// TIA Portal project "prova5arob" (V16)

(* hardware
DEVICE "S7-1200 station_1"  S7-1200 Station
   slot 0: "Telaio di montaggio_0"  S7-1200 Rack  Rack  V1.0
   slot 1: "PLC_1"  CPU 1215C DC/DC/Rly  6ES7 215-1HG40-0XB0  V4.2
DEVICE "HMI_1"  KTP700 Basic PN
   slot 0: "HMI_1"  KTP700 Basic PN  6AV2 123-2GB03-0AX0  16.0.0.0
   slot 1: "HMI_RT_1"  KTP700 Basic PN  6AV2 123-2GB03-0AX0  16.0.0.0
   slot 5: "HMI_1.IE_CP_1"  PROFINET Interface  16.0.0.0
      slot 1: "Interfaccia_1 PROFINET"  PROFINET Interface
         slot 1: "Porta_1"  Port
*)

// ===== PLC "PLC_1"  CPU 1215C DC/DC/Rly =====

DATA_BLOCK "Blocco_dati_pannello"   // DB1
{ S7_Optimized_Access := 'TRUE' }
VERSION : 0.1
   VAR
      Jog_start : Bool;
      spia_marcia : Bool;
   END_VAR
BEGIN
END_DATA_BLOCK

ORGANIZATION_BLOCK "Main"   // OB1, LAD, ProgramCycle
TITLE = "Main Program Sweep (Cycle)"
{ S7_Optimized_Access := 'TRUE' }
VERSION : 0.1
   VAR_INPUT
      Initial_Call : Bool;   // Initial call of this OB
      Remanence : Bool;   // =True, if remanent data are available
   END_VAR
BEGIN

REGION Network 1
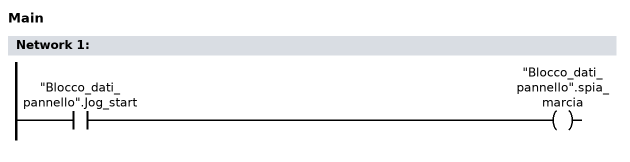
   RUNG wire#powerrail
      Contact( "Blocco_dati_pannello".Jog_start )
      Coil( "Blocco_dati_pannello".spia_marcia )
   END_RUNG
   // the same network as SCL:
   "Blocco_dati_pannello".spia_marcia := "Blocco_dati_pannello".Jog_start;
END_REGION
END_ORGANIZATION_BLOCK

(* ===== HMI "HMI_RT_1" =====
system functions are stored by id; their names below are inferred from use
connection "HMI_Collegamento_1": ETHERNET, SMART_S7_1200_OMS

HMI tags "Tabella delle variabili standard"
   "Variabile_Numero di pagina" : UInt, internal
   "Blocco_dati_pannello_Jog_start" : Bool = PLC Blocco_dati_pannello.Jog_start, 100 ms
   "Blocco_dati_pannello_spia_marcia" : Bool = PLC Blocco_dati_pannello.spia_marcia, 100 ms

text list "Elenco testi_Nome della pagina": 1 'Pagina base'

Template "Modello_1" 800x480
   Button "Esci" at 714,429 size 71x50; TextOff 'Esci'; PictureOff "ExitRuntime_KTP700_Basic_PN_TR"; PictureOn "ExitRuntime_KTP700_Basic_PN_TR"
      on Release: StopRuntime(0)
   Button "Template_Button" at 614,429 size 71x50; TextOff 'Text'
   Button "Template_Button_1" at 514,429 size 71x50; TextOff 'Text'
   Button "Template_Button_2" at 414,429 size 71x50; TextOff 'Text'
   Button "Template_Button_3" at 314,429 size 71x50; TextOff 'Text'
   Button "Template_Button_4" at 214,429 size 71x50; TextOff 'Text'
   Button "Template_Button_5" at 114,429 size 71x50; TextOff 'Text'
   Button "Pagina iniziale" at 14,429 size 71x50; TextOff 'Pagina iniziale'; PictureOff "NavigateHome_KTP700_Basic_PN_TR"; PictureOn "NavigateHome_KTP700_Basic_PN_TR"
      on Release: ActivateScreen("Pagina base", 0)
   SymbolicIOField "Pagina_campo_IO_simbolico" at 93,9 size 600x33; TextOff '0'; TextOn '1'; TextList "Elenco testi_Nome della pagina"
      ProcessValue <- "Variabile_Numero di pagina"
      on Change: ActivateScreenByNumber("Variabile_Numero di pagina", 0)
   DateTimeField "HmiScreenItemData" at 695,25 size 105x25
   DateTimeField "HmiScreenItemData_1" at 695,0 size 105x25
   GraphicView "Logo" at 0,0 size 91x51; Picture "Logo di HMI_1"

screen "Pagina base" 800x480, template "Modello_1"
   on GenerateScreen: SetTag("Variabile_Numero di pagina", 1)
   TextField "HmiScreenItemData" at 80,225 size 640x25; Text 'Benvenuto in HMI_1 (KTP700 Basic+ PN)!'
   Softkey "Softkey_F1" at 0,0 size 0x0
      on KeyDown: ActivateScreen("Pagina base", 0)
   Softkey "Softkey_F2" at 0,0 size 0x0
      on KeyDown: ActivateScreen("Pagina_1", 0)

screen "Pagina_1" 800x480
   Softkey "Softkey_F1" at 0,0 size 0x0
      on KeyDown: ActivateScreen("Pagina base", 0)
   Softkey "Softkey_F2" at 0,0 size 0x0
      on KeyDown: ActivateScreen("Pagina_1", 0)
   Button "FB_Right_Round" at 48,99 size 265x235; TextOff 'Text'; PictureOn "FB_Right_Round_Pressed_256c"; PictureOff "FB_Right_Round_Released_256c"
      on Press: SetBit("Blocco_dati_pannello_Jog_start")
      on Release: ResetBit("Blocco_dati_pannello_Jog_start")
   GraphicIOField "PlotLight_Round_G" at 366,114 size 216x215; PictureOn "PilotLight_Round_G_On_256c"; PictureOff "PilotLight_Round_G_Off_256c"
      ProcessValue <- "Blocco_dati_pannello_spia_marcia"
*)